// Pulses the selected RSR signal and waits for a fresh matching acknowledgement.
// Loss of bReady returns the FB to Idle without confirming the request.

FUNCTION_BLOCK FB_FanucStartProgram

VAR_INPUT
	bStart		: BOOL; // Rising edge starts a request while Idle and bReady; FALSE clears the FB error.
	nProgram	: INT; // Requested RSR selection, 1..8; latched when a valid request is accepted.
	bReady		: BOOL; // Enable permissive from FB_FanucEnable; must remain TRUE throughout the sequence.
	tAckTimeout	: TIME := T#2S; // Maximum additional wait for acknowledgement after the RSR pulse completes.
	stStatus	: ST_FanucStatus; // Live robot-status signals from FB_FanucStatus.
END_VAR

VAR_IN_OUT
	stControl	: ST_FanucControl; // Shared FANUC control structure; this FB writes Start_Program1..8 only.
END_VAR

VAR_OUTPUT
	bRequestActive	: BOOL; // TRUE while in Pulsing or WaitAck; does not indicate program execution.
	bDone			: BOOL; // TRUE for one PLC scan after the pulse completes and a fresh matching ACK is detected.
	bError			: BOOL; // TRUE in Error after invalid selection, ACK timeout, or invalid state; cleared by bStart = FALSE.
	eState			: E_FanucStartProgramState; // Current state exposed for diagnostics and HMI.
END_VAR

VAR
	eCurrentState	: E_FanucStartProgramState := E_FanucStartProgramState.Idle; // Internal state used by the sequence.
	rtStart			: R_TRIG; // Detects the FALSE-to-TRUE transition of bStart.
	nActiveProgram	: INT; // Latched RSR selection used for the active output and matching ACK.
	bActiveAck		: BOOL; // Current acknowledgement signal corresponding to nActiveProgram.
	bAckArmed		: BOOL; // TRUE once the selected ACK has been observed FALSE during the active sequence.
	bAckSeen		: BOOL; // Latched TRUE when the selected ACK is TRUE after acknowledgement detection is armed.
	bRsrPulseActive	: BOOL; // TRUE while the selected RSR output pulse is active.
	tonProgramPulse	: TON; // Measures the selected RSR pulse duration in Pulsing.
	tonAckTimeout	: TON; // Measures the additional acknowledgement wait in WaitAck.
END_VAR

VAR CONSTANT
	tProgramPulse : TIME := T#200MS; // Requested duration of the selected RSR output pulse on UI[9..16].
END_VAR

// Start edge detection
// ============================================================================
rtStart(CLK := bStart);

// Latch a valid program selection before reading its ACK
// ============================================================================
// This allows the Idle state to inspect the newly selected ACK before
// asserting the RSR output during this PLC scan.

IF (eCurrentState = E_FanucStartProgramState.Idle) AND rtStart.Q AND bReady AND (nProgram >= 1) AND (nProgram <= 8) THEN
	nActiveProgram := nProgram;
END_IF;


// Selected acknowledgement
// ============================================================================
CASE nActiveProgram OF

	1: bActiveAck := stStatus.bProg_Start1ACK;
	2: bActiveAck := stStatus.bProg_Start2ACK;
	3: bActiveAck := stStatus.bProg_Start3ACK;
	4: bActiveAck := stStatus.bProg_Start4ACK;
	5: bActiveAck := stStatus.bProg_Start5ACK;
	6: bActiveAck := stStatus.bProg_Start6ACK;
	7: bActiveAck := stStatus.bProg_Start7ACK;
	8: bActiveAck := stStatus.bProg_Start8ACK;

ELSE
	bActiveAck := FALSE;

END_CASE;


// Acknowledgement detection
// ============================================================================
// Remember a fresh ACK received during either the pulse or the ACK wait.
// An ACK already HIGH when the request is accepted must first become LOW.

IF (eCurrentState = E_FanucStartProgramState.Pulsing) OR (eCurrentState = E_FanucStartProgramState.WaitAck) THEN

	IF NOT bActiveAck THEN
		bAckArmed := TRUE;
	END_IF;

	IF bAckArmed AND bActiveAck THEN
		bAckSeen := TRUE;
	END_IF;

END_IF;

// State machine
// ============================================================================
CASE eCurrentState OF

	// IDLE
	// ========================================================================
	E_FanucStartProgramState.Idle:
	
		IF rtStart.Q AND bReady THEN
			IF (nProgram < 1) OR (nProgram > 8) THEN
				eCurrentState := E_FanucStartProgramState.Error;
			ELSE
				// nActiveProgram and its matching ACK were selected above.
				// Arm immediately if ACK is LOW before RSR is asserted.
				bAckArmed := NOT bActiveAck;
				bAckSeen := FALSE;

				eCurrentState := E_FanucStartProgramState.Pulsing;
			END_IF;
		END_IF;


	// PULSING
	// ========================================================================
	E_FanucStartProgramState.Pulsing:
	
		IF NOT bReady THEN
			eCurrentState := E_FanucStartProgramState.Idle;
		ELSIF tonProgramPulse.Q THEN
			// Complete the pulse even if ACK arrived before it ended.
			IF bAckSeen THEN
				eCurrentState := E_FanucStartProgramState.Done;
			ELSE
				eCurrentState := E_FanucStartProgramState.WaitAck;
			END_IF;
		END_IF;

	// WAIT FOR ACKNOWLEDGEMENT
	// ========================================================================
	E_FanucStartProgramState.WaitAck:

		IF NOT bReady THEN
			eCurrentState := E_FanucStartProgramState.Idle;
		ELSIF bAckSeen THEN
			eCurrentState := E_FanucStartProgramState.Done;
		ELSIF tonAckTimeout.Q THEN
			eCurrentState := E_FanucStartProgramState.Error;
		END_IF;

	// DONE
	// ========================================================================
	E_FanucStartProgramState.Done:

		// The Done state is exposed for one PLC scan.
		eCurrentState := E_FanucStartProgramState.Idle;

	// ERROR
	// ========================================================================
	E_FanucStartProgramState.Error:

		// Release Start before another request can be accepted.
		IF NOT bStart THEN
			eCurrentState := E_FanucStartProgramState.Idle;
		END_IF;

	// INVALID / UNKNOWN STATE
	// ========================================================================
	ELSE
		eCurrentState := E_FanucStartProgramState.Error;
END_CASE;


// Timers
// ============================================================================
// Each timer is called once per scan and enabled by its corresponding state.

tonProgramPulse(
	IN := (eCurrentState = E_FanucStartProgramState.Pulsing),
	PT := tProgramPulse
);

tonAckTimeout(
	IN := (eCurrentState = E_FanucStartProgramState.WaitAck),
	PT := tAckTimeout
);


// Clear handshake flags while Idle
// ============================================================================
IF eCurrentState = E_FanucStartProgramState.Idle THEN

	bAckArmed := FALSE;
	bAckSeen := FALSE;

END_IF;


// FANUC RSR control outputs
// ============================================================================
// Assign every RSR output once per scan.
// Only the selected output can be TRUE while the pulse is active.

bRsrPulseActive := (eCurrentState = E_FanucStartProgramState.Pulsing) AND NOT tonProgramPulse.Q;

stControl.Start_Program1 := bRsrPulseActive AND (nActiveProgram = 1);
stControl.Start_Program2 := bRsrPulseActive AND (nActiveProgram = 2);
stControl.Start_Program3 := bRsrPulseActive AND (nActiveProgram = 3);
stControl.Start_Program4 := bRsrPulseActive AND (nActiveProgram = 4);
stControl.Start_Program5 := bRsrPulseActive AND (nActiveProgram = 5);
stControl.Start_Program6 := bRsrPulseActive AND (nActiveProgram = 6);
stControl.Start_Program7 := bRsrPulseActive AND (nActiveProgram = 7);
stControl.Start_Program8 := bRsrPulseActive AND (nActiveProgram = 8);


// Diagnostic outputs
// ============================================================================
eState := eCurrentState;

bRequestActive := (eCurrentState = E_FanucStartProgramState.Pulsing) OR (eCurrentState = E_FanucStartProgramState.WaitAck);

bDone := (eCurrentState = E_FanucStartProgramState.Done);

bError := (eCurrentState = E_FanucStartProgramState.Error);

END_FUNCTION_BLOCK

(* stored: Version 1.1.0.1
   POU FB_FanucStartProgram: Id {639e9b5b-2378-78fc-0e0b-e22f6bfc1f16}, SpecialFunc None *)
